// SIMATIC S7-200 project (STEP 7-Micro/WIN), CPU 224 REL 02.01

ORGANIZATION_BLOCK Briquette_Press_A_V28:OB1
TITLE=A V2.8
// Custom program for WEIMA TH Standard Series briquette press.
//  #NVJOB Nicholas Veselov (independent developer) - https://nvjob.pro, http://nvjob.dx.am
BEGIN
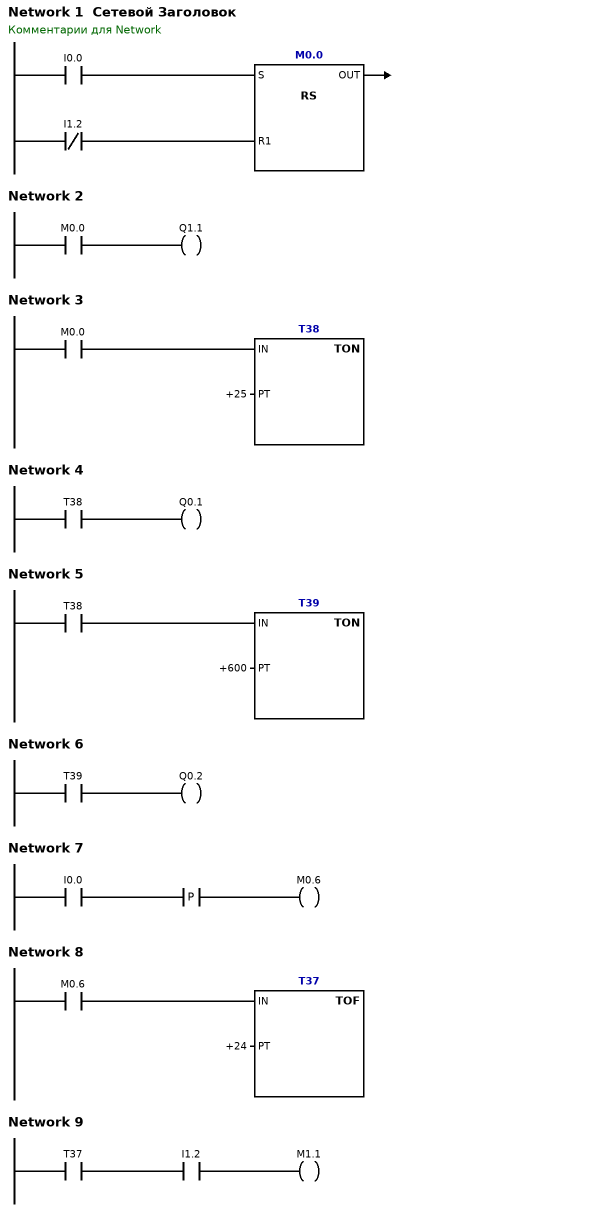
Network 1 // Сетевой Заголовок
// Комментарии для Network
LD     I0.0
LDN    I1.2
NOT
LPS
A      M0.0
=      M0.0
LPP
ALD
O      M0.0
=      M0.0
Network 2
LD     M0.0
=      Q1.1
Network 3
LD     M0.0
TON    T38, +25
Network 4
LD     T38
=      Q0.1
Network 5
LD     T38
TON    T39, +600
Network 6
LD     T39
=      Q0.2
Network 7
LD     I0.0
EU
=      M0.6
Network 8
LD     M0.6
TOF    T37, +24
Network 9
LD     T37
A      I1.2
=      M1.1
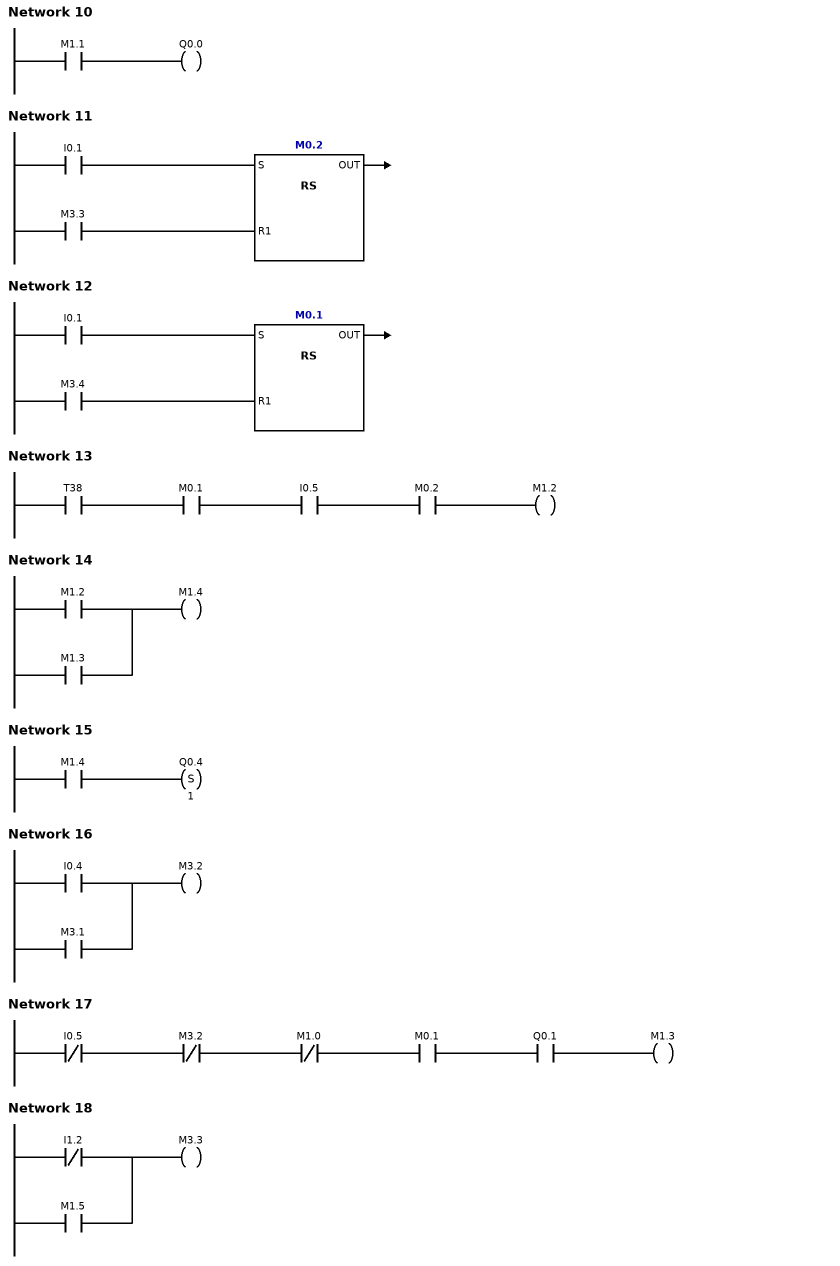
Network 10
LD     M1.1
=      Q0.0
Network 11
LD     I0.1
LD     M3.3
NOT
LPS
A      M0.2
=      M0.2
LPP
ALD
O      M0.2
=      M0.2
Network 12
LD     I0.1
LD     M3.4
NOT
LPS
A      M0.1
=      M0.1
LPP
ALD
O      M0.1
=      M0.1
Network 13
LD     T38
A      M0.1
A      I0.5
A      M0.2
=      M1.2
Network 14
LD     M1.2
O      M1.3
=      M1.4
Network 15
LD     M1.4
S      Q0.4, 1
Network 16
LD     I0.4
O      M3.1
=      M3.2
Network 17
LDN    I0.5
AN     M3.2
AN     M1.0
A      M0.1
A      Q0.1
=      M1.3
Network 18
LDN    I1.2
O      M1.5
=      M3.3
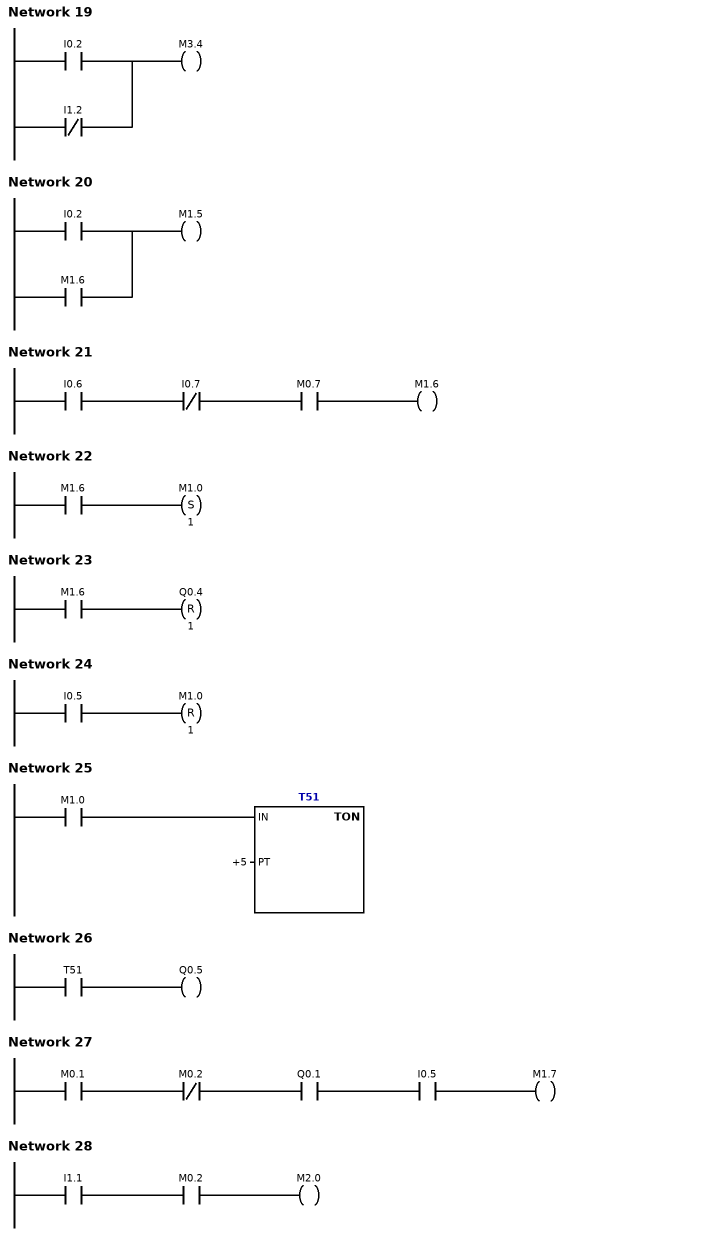
Network 19
LD     I0.2
ON     I1.2
=      M3.4
Network 20
LD     I0.2
O      M1.6
=      M1.5
Network 21
LD     I0.6
AN     I0.7
A      M0.7
=      M1.6
Network 22
LD     M1.6
S      M1.0, 1
Network 23
LD     M1.6
R      Q0.4, 1
Network 24
LD     I0.5
R      M1.0, 1
Network 25
LD     M1.0
TON    T51, +5
Network 26
LD     T51
=      Q0.5
Network 27
LD     M0.1
AN     M0.2
A      Q0.1
A      I0.5
=      M1.7
Network 28
LD     I1.1
A      M0.2
=      M2.0
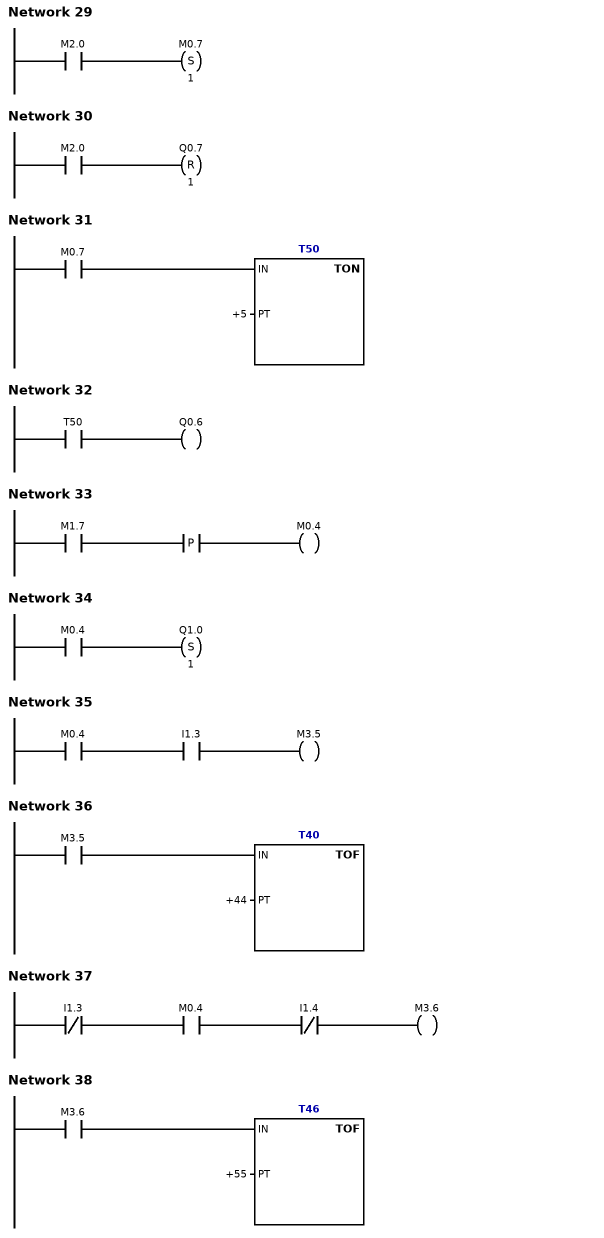
Network 29
LD     M2.0
S      M0.7, 1
Network 30
LD     M2.0
R      Q0.7, 1
Network 31
LD     M0.7
TON    T50, +5
Network 32
LD     T50
=      Q0.6
Network 33
LD     M1.7
EU
=      M0.4
Network 34
LD     M0.4
S      Q1.0, 1
Network 35
LD     M0.4
A      I1.3
=      M3.5
Network 36
LD     M3.5
TOF    T40, +44
Network 37
LDN    I1.3
A      M0.4
AN     I1.4
=      M3.6
Network 38
LD     M3.6
TOF    T46, +55
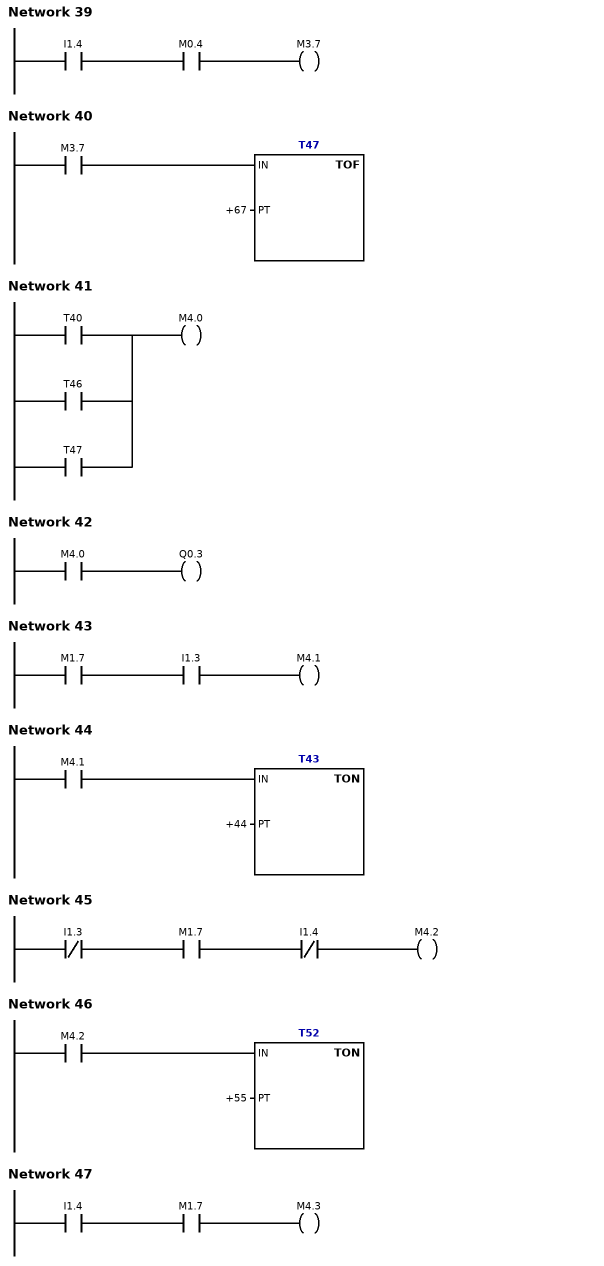
Network 39
LD     I1.4
A      M0.4
=      M3.7
Network 40
LD     M3.7
TOF    T47, +67
Network 41
LD     T40
O      T46
O      T47
=      M4.0
Network 42
LD     M4.0
=      Q0.3
Network 43
LD     M1.7
A      I1.3
=      M4.1
Network 44
LD     M4.1
TON    T43, +44
Network 45
LDN    I1.3
A      M1.7
AN     I1.4
=      M4.2
Network 46
LD     M4.2
TON    T52, +55
Network 47
LD     I1.4
A      M1.7
=      M4.3
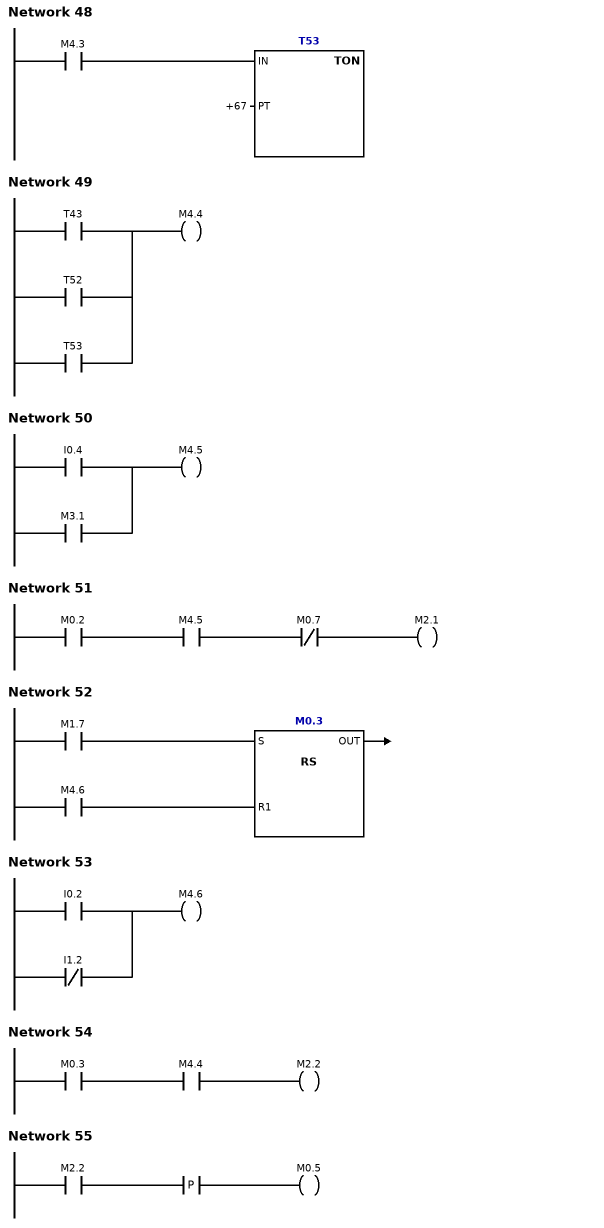
Network 48
LD     M4.3
TON    T53, +67
Network 49
LD     T43
O      T52
O      T53
=      M4.4
Network 50
LD     I0.4
O      M3.1
=      M4.5
Network 51
LD     M0.2
A      M4.5
AN     M0.7
=      M2.1
Network 52
LD     M1.7
LD     M4.6
NOT
LPS
A      M0.3
=      M0.3
LPP
ALD
O      M0.3
=      M0.3
Network 53
LD     I0.2
ON     I1.2
=      M4.6
Network 54
LD     M0.3
A      M4.4
=      M2.2
Network 55
LD     M2.2
EU
=      M0.5
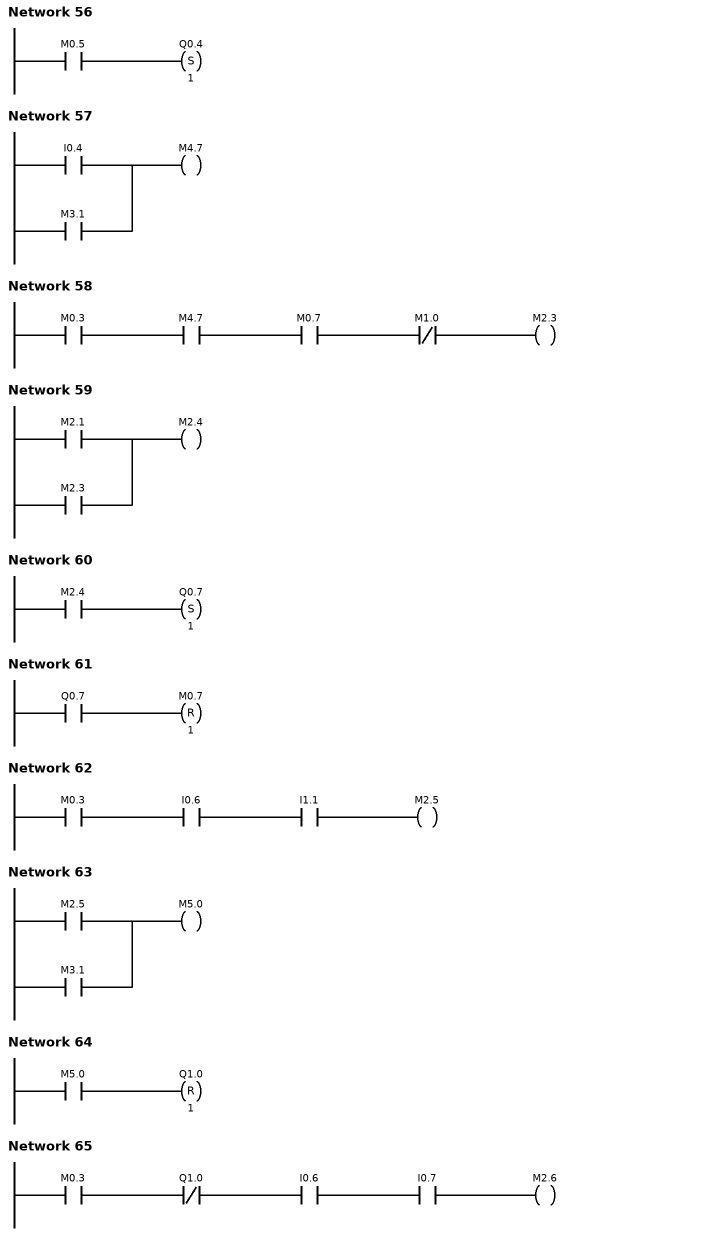
Network 56
LD     M0.5
S      Q0.4, 1
Network 57
LD     I0.4
O      M3.1
=      M4.7
Network 58
LD     M0.3
A      M4.7
A      M0.7
AN     M1.0
=      M2.3
Network 59
LD     M2.1
O      M2.3
=      M2.4
Network 60
LD     M2.4
S      Q0.7, 1
Network 61
LD     Q0.7
R      M0.7, 1
Network 62
LD     M0.3
A      I0.6
A      I1.1
=      M2.5
Network 63
LD     M2.5
O      M3.1
=      M5.0
Network 64
LD     M5.0
R      Q1.0, 1
Network 65
LD     M0.3
AN     Q1.0
A      I0.6
A      I0.7
=      M2.6
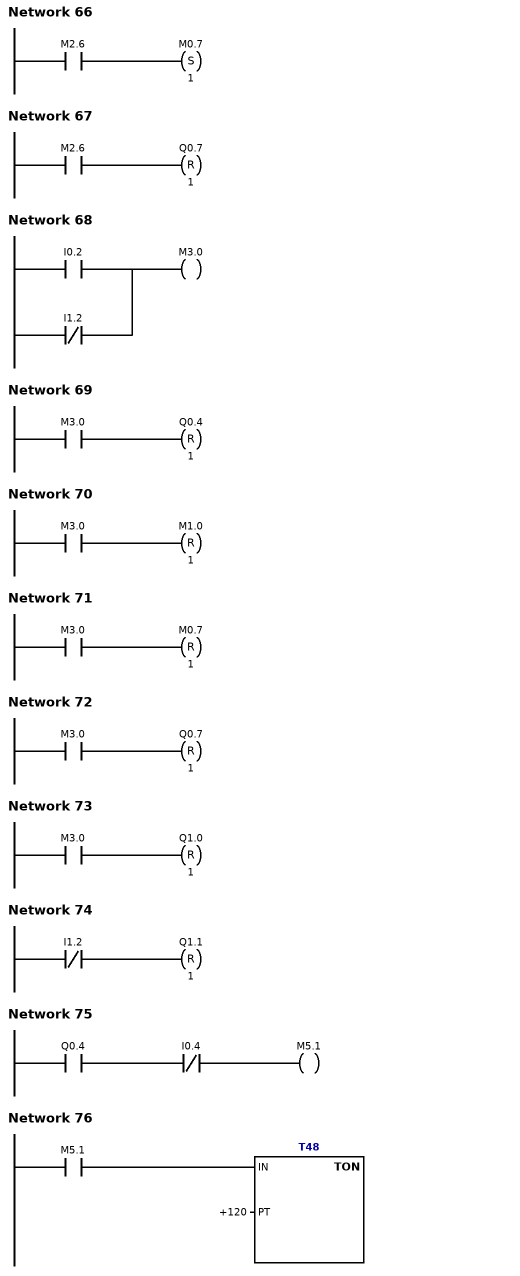
Network 66
LD     M2.6
S      M0.7, 1
Network 67
LD     M2.6
R      Q0.7, 1
Network 68
LD     I0.2
ON     I1.2
=      M3.0
Network 69
LD     M3.0
R      Q0.4, 1
Network 70
LD     M3.0
R      M1.0, 1
Network 71
LD     M3.0
R      M0.7, 1
Network 72
LD     M3.0
R      Q0.7, 1
Network 73
LD     M3.0
R      Q1.0, 1
Network 74
LDN    I1.2
R      Q1.1, 1
Network 75
LD     Q0.4
AN     I0.4
=      M5.1
Network 76
LD     M5.1
TON    T48, +120
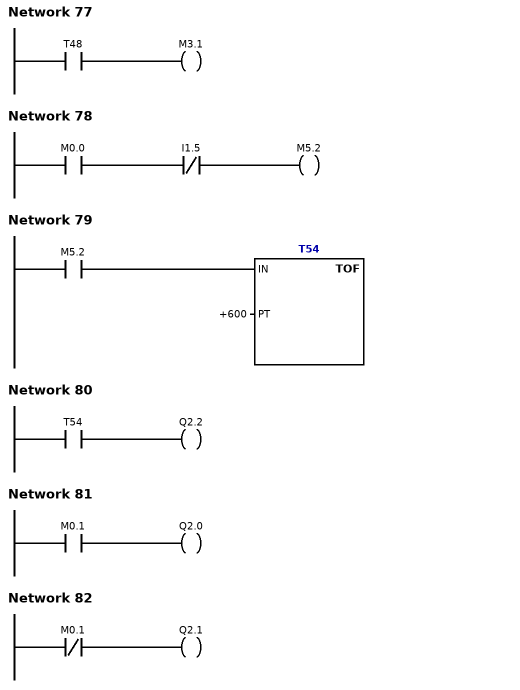
Network 77
LD     T48
=      M3.1
Network 78
LD     M0.0
AN     I1.5
=      M5.2
Network 79
LD     M5.2
TOF    T54, +600
Network 80
LD     T54
=      Q2.2
Network 81
LD     M0.1
=      Q2.0
Network 82
LDN    M0.1
=      Q2.1
END_ORGANIZATION_BLOCK
